REGION Network 97: Step[2046] : Tape Attach Unit HomePos Command
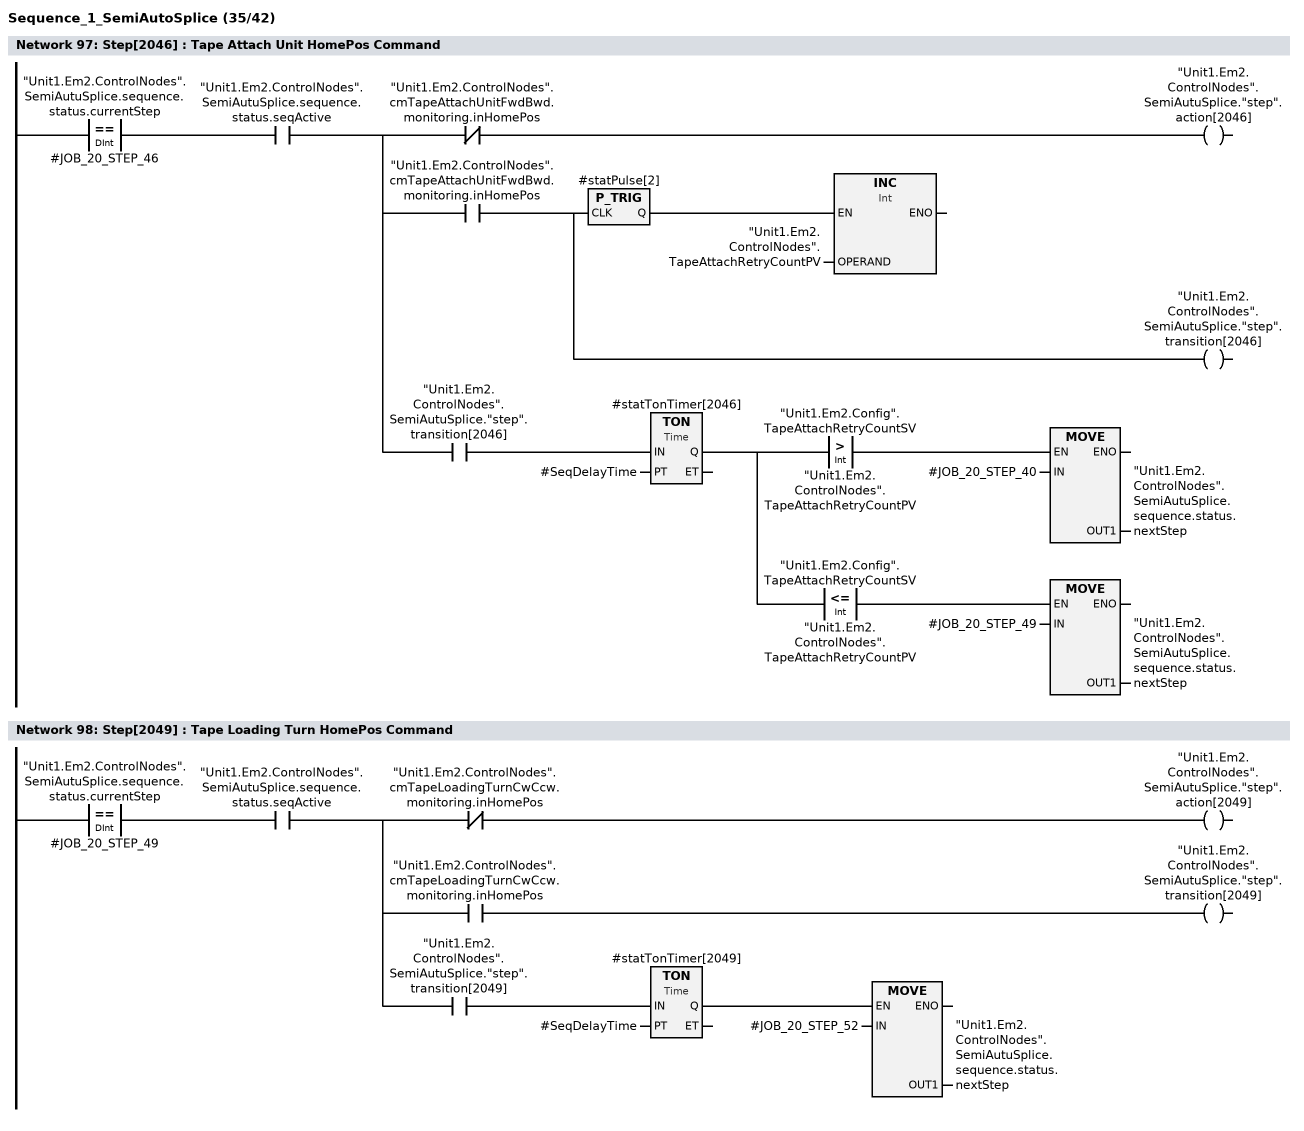
   RUNG wire#powerrail
      { S7_Templates := "SrcType := DInt" } EQ_Contact(in1 := "Unit1.Em2.ControlNodes".SemiAutuSplice.sequence.status.currentStep, in2 := #JOB_20_STEP_46)
      Contact( "Unit1.Em2.ControlNodes".SemiAutuSplice.sequence.status.seqActive )
      wire#w1
      I_Contact( "Unit1.Em2.ControlNodes".cmTapeAttachUnitFwdBwd.monitoring.inHomePos )
      Coil( "Unit1.Em2.ControlNodes".SemiAutuSplice."step".action[2046] )
   END_RUNG
   RUNG wire#w1
      Contact( "Unit1.Em2.ControlNodes".cmTapeAttachUnitFwdBwd.monitoring.inHomePos )
      wire#w2
      P_Trig( #statPulse[2] )
      { S7_Templates := "DestType := Int" } Inc( "Unit1.Em2.ControlNodes".TapeAttachRetryCountPV )
   END_RUNG
   RUNG wire#w2
      Coil( "Unit1.Em2.ControlNodes".SemiAutuSplice."step".transition[2046] )
   END_RUNG
   RUNG wire#w1
      Contact( "Unit1.Em2.ControlNodes".SemiAutuSplice."step".transition[2046] )
      { S7_Templates := "time_type := Time" } #statTonTimer[2046].TON(pt := #SeqDelayTime, et =>)
      wire#w3
      { S7_Templates := "SrcType := Int" } GT_Contact(in1 := "Unit1.Em2.Config".TapeAttachRetryCountSV, in2 := "Unit1.Em2.ControlNodes".TapeAttachRetryCountPV)
      Move(in := #JOB_20_STEP_40, out1 => "Unit1.Em2.ControlNodes".SemiAutuSplice.sequence.status.nextStep)
   END_RUNG
   RUNG wire#w3
      { S7_Templates := "SrcType := Int" } LE_Contact(in1 := "Unit1.Em2.Config".TapeAttachRetryCountSV, in2 := "Unit1.Em2.ControlNodes".TapeAttachRetryCountPV)
      Move(in := #JOB_20_STEP_49, out1 => "Unit1.Em2.ControlNodes".SemiAutuSplice.sequence.status.nextStep)
   END_RUNG
   // the same network as SCL:
   #_w1 := ("Unit1.Em2.ControlNodes".SemiAutuSplice.sequence.status.currentStep = #JOB_20_STEP_46) AND "Unit1.Em2.ControlNodes".SemiAutuSplice.sequence.status.seqActive;
   "Unit1.Em2.ControlNodes".SemiAutuSplice."step".action[2046] := #_w1 AND NOT "Unit1.Em2.ControlNodes".cmTapeAttachUnitFwdBwd.monitoring.inHomePos;
   #_w2 := #_w1 AND "Unit1.Em2.ControlNodes".cmTapeAttachUnitFwdBwd.monitoring.inHomePos;
   #_w3 := #_w2 AND NOT #statPulse[2];   // rising edge
   #statPulse[2] := #_w2;
   IF #_w3 THEN
       "Unit1.Em2.ControlNodes".TapeAttachRetryCountPV := "Unit1.Em2.ControlNodes".TapeAttachRetryCountPV + 1;
   END_IF;
   "Unit1.Em2.ControlNodes".SemiAutuSplice."step".transition[2046] := #_w2;
   #statTonTimer[2046].TON(IN := #_w1 AND "Unit1.Em2.ControlNodes".SemiAutuSplice."step".transition[2046],
                           PT := #SeqDelayTime);
   IF #statTonTimer[2046].Q AND ("Unit1.Em2.Config".TapeAttachRetryCountSV > "Unit1.Em2.ControlNodes".TapeAttachRetryCountPV) THEN
       "Unit1.Em2.ControlNodes".SemiAutuSplice.sequence.status.nextStep := #JOB_20_STEP_40;
   END_IF;
   IF #statTonTimer[2046].Q AND ("Unit1.Em2.Config".TapeAttachRetryCountSV <= "Unit1.Em2.ControlNodes".TapeAttachRetryCountPV) THEN
       "Unit1.Em2.ControlNodes".SemiAutuSplice.sequence.status.nextStep := #JOB_20_STEP_49;
   END_IF;
END_REGION

REGION Network 98: Step[2049] : Tape Loading Turn HomePos Command
   RUNG wire#powerrail
      { S7_Templates := "SrcType := DInt" } EQ_Contact(in1 := "Unit1.Em2.ControlNodes".SemiAutuSplice.sequence.status.currentStep, in2 := #JOB_20_STEP_49)
      Contact( "Unit1.Em2.ControlNodes".SemiAutuSplice.sequence.status.seqActive )
      wire#w1
      I_Contact( "Unit1.Em2.ControlNodes".cmTapeLoadingTurnCwCcw.monitoring.inHomePos )
      Coil( "Unit1.Em2.ControlNodes".SemiAutuSplice."step".action[2049] )
   END_RUNG
   RUNG wire#w1
      Contact( "Unit1.Em2.ControlNodes".cmTapeLoadingTurnCwCcw.monitoring.inHomePos )
      Coil( "Unit1.Em2.ControlNodes".SemiAutuSplice."step".transition[2049] )
   END_RUNG
   RUNG wire#w1
      Contact( "Unit1.Em2.ControlNodes".SemiAutuSplice."step".transition[2049] )
      { S7_Templates := "time_type := Time" } #statTonTimer[2049].TON(pt := #SeqDelayTime, et =>)
      Move(in := #JOB_20_STEP_52, out1 => "Unit1.Em2.ControlNodes".SemiAutuSplice.sequence.status.nextStep)
   END_RUNG
   // the same network as SCL:
   #_w1 := ("Unit1.Em2.ControlNodes".SemiAutuSplice.sequence.status.currentStep = #JOB_20_STEP_49) AND "Unit1.Em2.ControlNodes".SemiAutuSplice.sequence.status.seqActive;
   "Unit1.Em2.ControlNodes".SemiAutuSplice."step".action[2049] := #_w1 AND NOT "Unit1.Em2.ControlNodes".cmTapeLoadingTurnCwCcw.monitoring.inHomePos;
   "Unit1.Em2.ControlNodes".SemiAutuSplice."step".transition[2049] := #_w1 AND "Unit1.Em2.ControlNodes".cmTapeLoadingTurnCwCcw.monitoring.inHomePos;
   #statTonTimer[2049].TON(IN := #_w1 AND "Unit1.Em2.ControlNodes".SemiAutuSplice."step".transition[2049],
                           PT := #SeqDelayTime);
   IF #statTonTimer[2049].Q THEN
       "Unit1.Em2.ControlNodes".SemiAutuSplice.sequence.status.nextStep := #JOB_20_STEP_52;
   END_IF;
END_REGION

REGION Network 99: Step[2052] : Uw Semi Splicer Vacuum Top & Uw Semi Splicer Vacuum Bottom HomePos Command
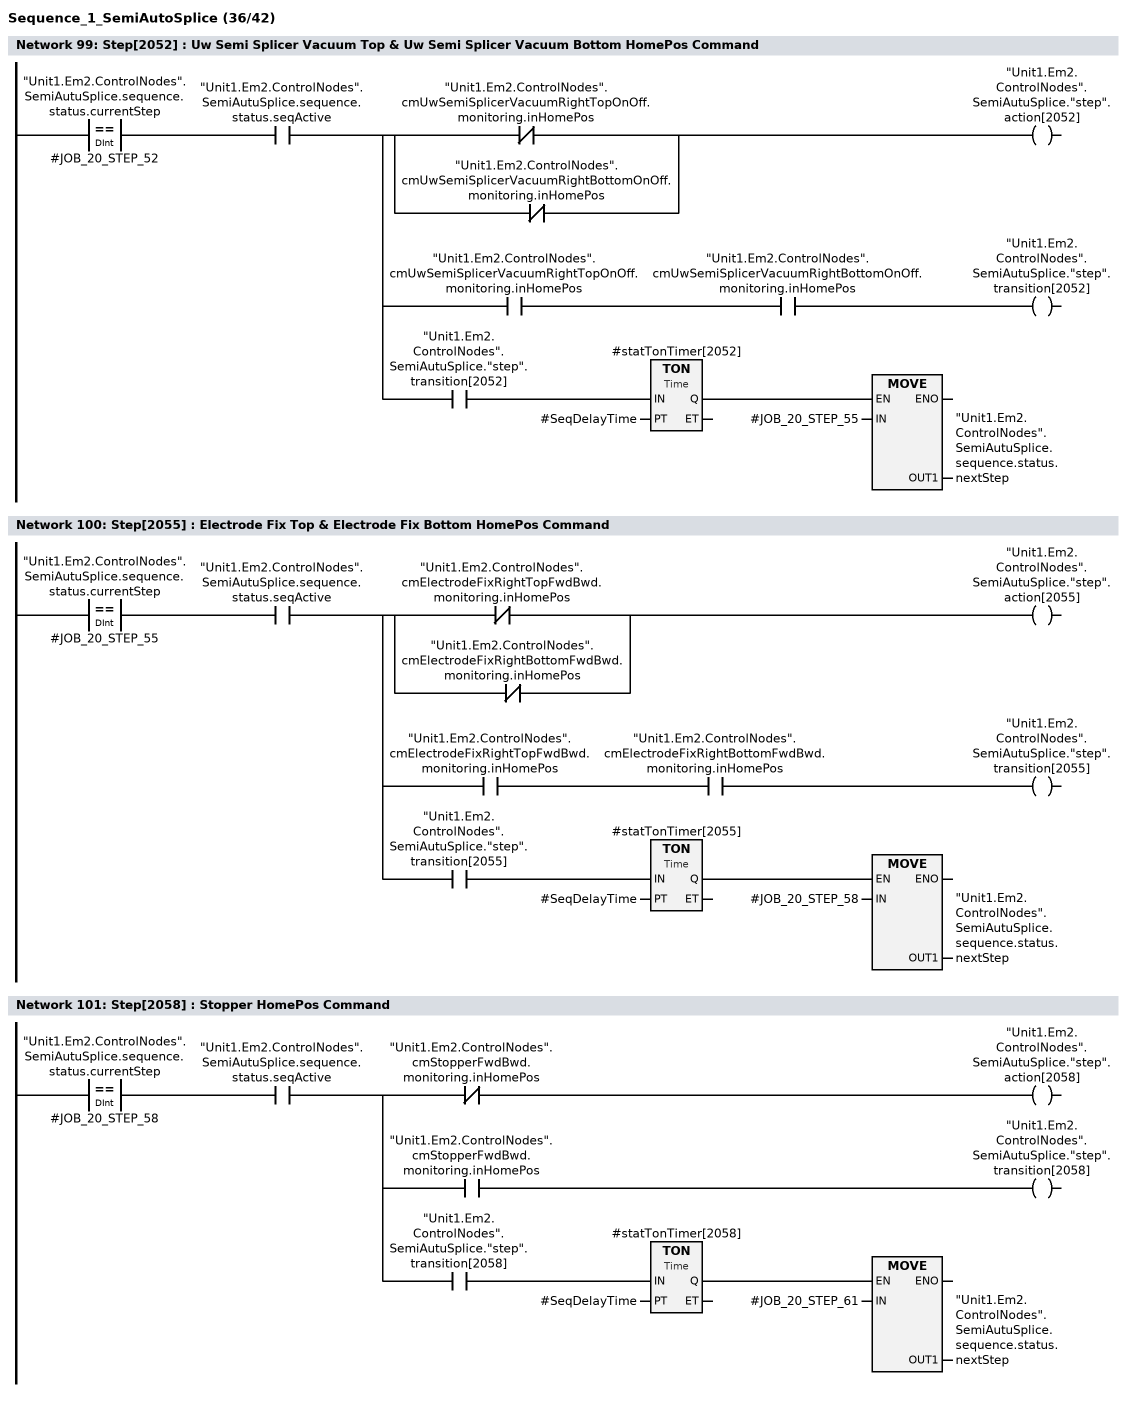
   RUNG wire#powerrail
      { S7_Templates := "SrcType := DInt" } EQ_Contact(in1 := "Unit1.Em2.ControlNodes".SemiAutuSplice.sequence.status.currentStep, in2 := #JOB_20_STEP_52)
      Contact( "Unit1.Em2.ControlNodes".SemiAutuSplice.sequence.status.seqActive )
      wire#w1
      I_Contact( "Unit1.Em2.ControlNodes".cmUwSemiSplicerVacuumRightTopOnOff.monitoring.inHomePos )
      wire#w2
      Coil( "Unit1.Em2.ControlNodes".SemiAutuSplice."step".action[2052] )
   END_RUNG
   RUNG wire#w1
      I_Contact( "Unit1.Em2.ControlNodes".cmUwSemiSplicerVacuumRightBottomOnOff.monitoring.inHomePos )
   END_RUNG wire#w2
   RUNG wire#w1
      Contact( "Unit1.Em2.ControlNodes".cmUwSemiSplicerVacuumRightTopOnOff.monitoring.inHomePos )
      Contact( "Unit1.Em2.ControlNodes".cmUwSemiSplicerVacuumRightBottomOnOff.monitoring.inHomePos )
      Coil( "Unit1.Em2.ControlNodes".SemiAutuSplice."step".transition[2052] )
   END_RUNG
   RUNG wire#w1
      Contact( "Unit1.Em2.ControlNodes".SemiAutuSplice."step".transition[2052] )
      { S7_Templates := "time_type := Time" } #statTonTimer[2052].TON(pt := #SeqDelayTime, et =>)
      Move(in := #JOB_20_STEP_55, out1 => "Unit1.Em2.ControlNodes".SemiAutuSplice.sequence.status.nextStep)
   END_RUNG
   // the same network as SCL:
   #_w1 := ("Unit1.Em2.ControlNodes".SemiAutuSplice.sequence.status.currentStep = #JOB_20_STEP_52) AND "Unit1.Em2.ControlNodes".SemiAutuSplice.sequence.status.seqActive;
   "Unit1.Em2.ControlNodes".SemiAutuSplice."step".action[2052] := #_w1 AND (NOT "Unit1.Em2.ControlNodes".cmUwSemiSplicerVacuumRightTopOnOff.monitoring.inHomePos OR NOT "Unit1.Em2.ControlNodes".cmUwSemiSplicerVacuumRightBottomOnOff.monitoring.inHomePos);
   "Unit1.Em2.ControlNodes".SemiAutuSplice."step".transition[2052] := #_w1 AND "Unit1.Em2.ControlNodes".cmUwSemiSplicerVacuumRightTopOnOff.monitoring.inHomePos AND "Unit1.Em2.ControlNodes".cmUwSemiSplicerVacuumRightBottomOnOff.monitoring.inHomePos;
   #statTonTimer[2052].TON(IN := #_w1 AND "Unit1.Em2.ControlNodes".SemiAutuSplice."step".transition[2052],
                           PT := #SeqDelayTime);
   IF #statTonTimer[2052].Q THEN
       "Unit1.Em2.ControlNodes".SemiAutuSplice.sequence.status.nextStep := #JOB_20_STEP_55;
   END_IF;
END_REGION

REGION Network 100: Step[2055] : Electrode Fix Top & Electrode Fix Bottom HomePos Command
   RUNG wire#powerrail
      { S7_Templates := "SrcType := DInt" } EQ_Contact(in1 := "Unit1.Em2.ControlNodes".SemiAutuSplice.sequence.status.currentStep, in2 := #JOB_20_STEP_55)
      Contact( "Unit1.Em2.ControlNodes".SemiAutuSplice.sequence.status.seqActive )
      wire#w1
      I_Contact( "Unit1.Em2.ControlNodes".cmElectrodeFixRightTopFwdBwd.monitoring.inHomePos )
      wire#w2
      Coil( "Unit1.Em2.ControlNodes".SemiAutuSplice."step".action[2055] )
   END_RUNG
   RUNG wire#w1
      I_Contact( "Unit1.Em2.ControlNodes".cmElectrodeFixRightBottomFwdBwd.monitoring.inHomePos )
   END_RUNG wire#w2
   RUNG wire#w1
      Contact( "Unit1.Em2.ControlNodes".cmElectrodeFixRightTopFwdBwd.monitoring.inHomePos )
      Contact( "Unit1.Em2.ControlNodes".cmElectrodeFixRightBottomFwdBwd.monitoring.inHomePos )
      Coil( "Unit1.Em2.ControlNodes".SemiAutuSplice."step".transition[2055] )
   END_RUNG
   RUNG wire#w1
      Contact( "Unit1.Em2.ControlNodes".SemiAutuSplice."step".transition[2055] )
      { S7_Templates := "time_type := Time" } #statTonTimer[2055].TON(pt := #SeqDelayTime, et =>)
      Move(in := #JOB_20_STEP_58, out1 => "Unit1.Em2.ControlNodes".SemiAutuSplice.sequence.status.nextStep)
   END_RUNG
   // the same network as SCL:
   #_w1 := ("Unit1.Em2.ControlNodes".SemiAutuSplice.sequence.status.currentStep = #JOB_20_STEP_55) AND "Unit1.Em2.ControlNodes".SemiAutuSplice.sequence.status.seqActive;
   "Unit1.Em2.ControlNodes".SemiAutuSplice."step".action[2055] := #_w1 AND (NOT "Unit1.Em2.ControlNodes".cmElectrodeFixRightTopFwdBwd.monitoring.inHomePos OR NOT "Unit1.Em2.ControlNodes".cmElectrodeFixRightBottomFwdBwd.monitoring.inHomePos);
   "Unit1.Em2.ControlNodes".SemiAutuSplice."step".transition[2055] := #_w1 AND "Unit1.Em2.ControlNodes".cmElectrodeFixRightTopFwdBwd.monitoring.inHomePos AND "Unit1.Em2.ControlNodes".cmElectrodeFixRightBottomFwdBwd.monitoring.inHomePos;
   #statTonTimer[2055].TON(IN := #_w1 AND "Unit1.Em2.ControlNodes".SemiAutuSplice."step".transition[2055],
                           PT := #SeqDelayTime);
   IF #statTonTimer[2055].Q THEN
       "Unit1.Em2.ControlNodes".SemiAutuSplice.sequence.status.nextStep := #JOB_20_STEP_58;
   END_IF;
END_REGION

REGION Network 101: Step[2058] : Stopper HomePos Command
   RUNG wire#powerrail
      { S7_Templates := "SrcType := DInt" } EQ_Contact(in1 := "Unit1.Em2.ControlNodes".SemiAutuSplice.sequence.status.currentStep, in2 := #JOB_20_STEP_58)
      Contact( "Unit1.Em2.ControlNodes".SemiAutuSplice.sequence.status.seqActive )
      wire#w1
      I_Contact( "Unit1.Em2.ControlNodes".cmStopperFwdBwd.monitoring.inHomePos )
      Coil( "Unit1.Em2.ControlNodes".SemiAutuSplice."step".action[2058] )
   END_RUNG
   RUNG wire#w1
      Contact( "Unit1.Em2.ControlNodes".cmStopperFwdBwd.monitoring.inHomePos )
      Coil( "Unit1.Em2.ControlNodes".SemiAutuSplice."step".transition[2058] )
   END_RUNG
   RUNG wire#w1
      Contact( "Unit1.Em2.ControlNodes".SemiAutuSplice."step".transition[2058] )
      { S7_Templates := "time_type := Time" } #statTonTimer[2058].TON(pt := #SeqDelayTime, et =>)
      Move(in := #JOB_20_STEP_61, out1 => "Unit1.Em2.ControlNodes".SemiAutuSplice.sequence.status.nextStep)
   END_RUNG
   // the same network as SCL:
   #_w1 := ("Unit1.Em2.ControlNodes".SemiAutuSplice.sequence.status.currentStep = #JOB_20_STEP_58) AND "Unit1.Em2.ControlNodes".SemiAutuSplice.sequence.status.seqActive;
   "Unit1.Em2.ControlNodes".SemiAutuSplice."step".action[2058] := #_w1 AND NOT "Unit1.Em2.ControlNodes".cmStopperFwdBwd.monitoring.inHomePos;
   "Unit1.Em2.ControlNodes".SemiAutuSplice."step".transition[2058] := #_w1 AND "Unit1.Em2.ControlNodes".cmStopperFwdBwd.monitoring.inHomePos;
   #statTonTimer[2058].TON(IN := #_w1 AND "Unit1.Em2.ControlNodes".SemiAutuSplice."step".transition[2058],
                           PT := #SeqDelayTime);
   IF #statTonTimer[2058].Q THEN
       "Unit1.Em2.ControlNodes".SemiAutuSplice.sequence.status.nextStep := #JOB_20_STEP_61;
   END_IF;
END_REGION

REGION Network 102: Step[2061] : EM Link Change Check
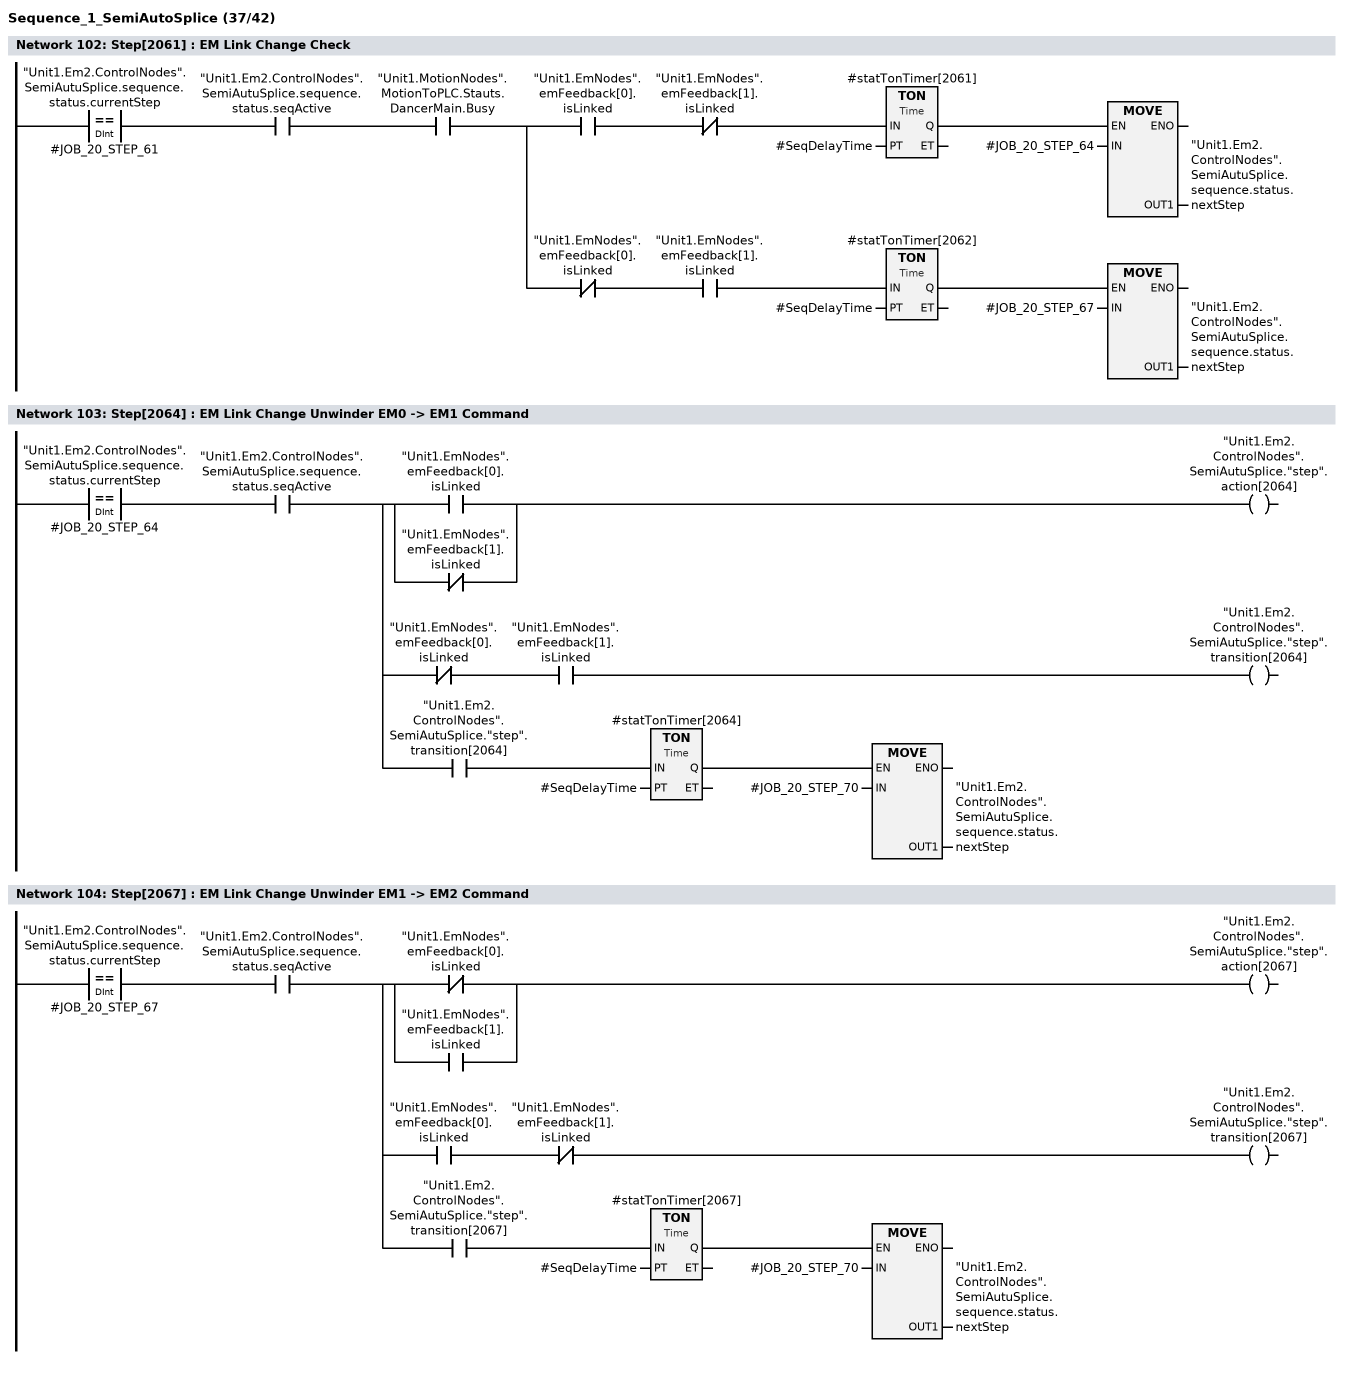
   RUNG wire#powerrail
      { S7_Templates := "SrcType := DInt" } EQ_Contact(in1 := "Unit1.Em2.ControlNodes".SemiAutuSplice.sequence.status.currentStep, in2 := #JOB_20_STEP_61)
      Contact( "Unit1.Em2.ControlNodes".SemiAutuSplice.sequence.status.seqActive )
      Contact( "Unit1.MotionNodes".MotionToPLC.Stauts.DancerMain.Busy )
      wire#w1
      Contact( "Unit1.EmNodes".emFeedback[0].isLinked )
      I_Contact( "Unit1.EmNodes".emFeedback[1].isLinked )
      { S7_Templates := "time_type := Time" } #statTonTimer[2061].TON(pt := #SeqDelayTime, et =>)
      Move(in := #JOB_20_STEP_64, out1 => "Unit1.Em2.ControlNodes".SemiAutuSplice.sequence.status.nextStep)
   END_RUNG
   RUNG wire#w1
      I_Contact( "Unit1.EmNodes".emFeedback[0].isLinked )
      Contact( "Unit1.EmNodes".emFeedback[1].isLinked )
      { S7_Templates := "time_type := Time" } #statTonTimer[2062].TON(pt := #SeqDelayTime, et =>)
      Move(in := #JOB_20_STEP_67, out1 => "Unit1.Em2.ControlNodes".SemiAutuSplice.sequence.status.nextStep)
   END_RUNG
   // the same network as SCL:
   #_w1 := ("Unit1.Em2.ControlNodes".SemiAutuSplice.sequence.status.currentStep = #JOB_20_STEP_61) AND "Unit1.Em2.ControlNodes".SemiAutuSplice.sequence.status.seqActive AND "Unit1.MotionNodes".MotionToPLC.Stauts.DancerMain.Busy;
   #statTonTimer[2061].TON(IN := #_w1 AND "Unit1.EmNodes".emFeedback[0].isLinked AND NOT "Unit1.EmNodes".emFeedback[1].isLinked,
                           PT := #SeqDelayTime);
   IF #statTonTimer[2061].Q THEN
       "Unit1.Em2.ControlNodes".SemiAutuSplice.sequence.status.nextStep := #JOB_20_STEP_64;
   END_IF;
   #statTonTimer[2062].TON(IN := #_w1 AND NOT "Unit1.EmNodes".emFeedback[0].isLinked AND "Unit1.EmNodes".emFeedback[1].isLinked,
                           PT := #SeqDelayTime);
   IF #statTonTimer[2062].Q THEN
       "Unit1.Em2.ControlNodes".SemiAutuSplice.sequence.status.nextStep := #JOB_20_STEP_67;
   END_IF;
END_REGION

REGION Network 103: Step[2064] : EM Link Change Unwinder EM0 -> EM1 Command
   RUNG wire#powerrail
      { S7_Templates := "SrcType := DInt" } EQ_Contact(in1 := "Unit1.Em2.ControlNodes".SemiAutuSplice.sequence.status.currentStep, in2 := #JOB_20_STEP_64)
      Contact( "Unit1.Em2.ControlNodes".SemiAutuSplice.sequence.status.seqActive )
      wire#w1
      Contact( "Unit1.EmNodes".emFeedback[0].isLinked )
      wire#w2
      Coil( "Unit1.Em2.ControlNodes".SemiAutuSplice."step".action[2064] )
   END_RUNG
   RUNG wire#w1
      I_Contact( "Unit1.EmNodes".emFeedback[1].isLinked )
   END_RUNG wire#w2
   RUNG wire#w1
      I_Contact( "Unit1.EmNodes".emFeedback[0].isLinked )
      Contact( "Unit1.EmNodes".emFeedback[1].isLinked )
      Coil( "Unit1.Em2.ControlNodes".SemiAutuSplice."step".transition[2064] )
   END_RUNG
   RUNG wire#w1
      Contact( "Unit1.Em2.ControlNodes".SemiAutuSplice."step".transition[2064] )
      { S7_Templates := "time_type := Time" } #statTonTimer[2064].TON(pt := #SeqDelayTime, et =>)
      Move(in := #JOB_20_STEP_70, out1 => "Unit1.Em2.ControlNodes".SemiAutuSplice.sequence.status.nextStep)
   END_RUNG
   // the same network as SCL:
   #_w1 := ("Unit1.Em2.ControlNodes".SemiAutuSplice.sequence.status.currentStep = #JOB_20_STEP_64) AND "Unit1.Em2.ControlNodes".SemiAutuSplice.sequence.status.seqActive;
   "Unit1.Em2.ControlNodes".SemiAutuSplice."step".action[2064] := #_w1 AND ("Unit1.EmNodes".emFeedback[0].isLinked OR NOT "Unit1.EmNodes".emFeedback[1].isLinked);
   "Unit1.Em2.ControlNodes".SemiAutuSplice."step".transition[2064] := #_w1 AND NOT "Unit1.EmNodes".emFeedback[0].isLinked AND "Unit1.EmNodes".emFeedback[1].isLinked;
   #statTonTimer[2064].TON(IN := #_w1 AND "Unit1.Em2.ControlNodes".SemiAutuSplice."step".transition[2064],
                           PT := #SeqDelayTime);
   IF #statTonTimer[2064].Q THEN
       "Unit1.Em2.ControlNodes".SemiAutuSplice.sequence.status.nextStep := #JOB_20_STEP_70;
   END_IF;
END_REGION

REGION Network 104: Step[2067] : EM Link Change Unwinder EM1 -> EM2 Command
   RUNG wire#powerrail
      { S7_Templates := "SrcType := DInt" } EQ_Contact(in1 := "Unit1.Em2.ControlNodes".SemiAutuSplice.sequence.status.currentStep, in2 := #JOB_20_STEP_67)
      Contact( "Unit1.Em2.ControlNodes".SemiAutuSplice.sequence.status.seqActive )
      wire#w1
      I_Contact( "Unit1.EmNodes".emFeedback[0].isLinked )
      wire#w2
      Coil( "Unit1.Em2.ControlNodes".SemiAutuSplice."step".action[2067] )
   END_RUNG
   RUNG wire#w1
      Contact( "Unit1.EmNodes".emFeedback[1].isLinked )
   END_RUNG wire#w2
   RUNG wire#w1
      Contact( "Unit1.EmNodes".emFeedback[0].isLinked )
      I_Contact( "Unit1.EmNodes".emFeedback[1].isLinked )
      Coil( "Unit1.Em2.ControlNodes".SemiAutuSplice."step".transition[2067] )
   END_RUNG
   RUNG wire#w1
      Contact( "Unit1.Em2.ControlNodes".SemiAutuSplice."step".transition[2067] )
      { S7_Templates := "time_type := Time" } #statTonTimer[2067].TON(pt := #SeqDelayTime, et =>)
      Move(in := #JOB_20_STEP_70, out1 => "Unit1.Em2.ControlNodes".SemiAutuSplice.sequence.status.nextStep)
   END_RUNG
   // the same network as SCL:
   #_w1 := ("Unit1.Em2.ControlNodes".SemiAutuSplice.sequence.status.currentStep = #JOB_20_STEP_67) AND "Unit1.Em2.ControlNodes".SemiAutuSplice.sequence.status.seqActive;
   "Unit1.Em2.ControlNodes".SemiAutuSplice."step".action[2067] := #_w1 AND (NOT "Unit1.EmNodes".emFeedback[0].isLinked OR "Unit1.EmNodes".emFeedback[1].isLinked);
   "Unit1.Em2.ControlNodes".SemiAutuSplice."step".transition[2067] := #_w1 AND "Unit1.EmNodes".emFeedback[0].isLinked AND NOT "Unit1.EmNodes".emFeedback[1].isLinked;
   #statTonTimer[2067].TON(IN := #_w1 AND "Unit1.Em2.ControlNodes".SemiAutuSplice."step".transition[2067],
                           PT := #SeqDelayTime);
   IF #statTonTimer[2067].Q THEN
       "Unit1.Em2.ControlNodes".SemiAutuSplice.sequence.status.nextStep := #JOB_20_STEP_70;
   END_IF;
END_REGION

REGION Network 105: Step[2070] : EM Link Change Comp
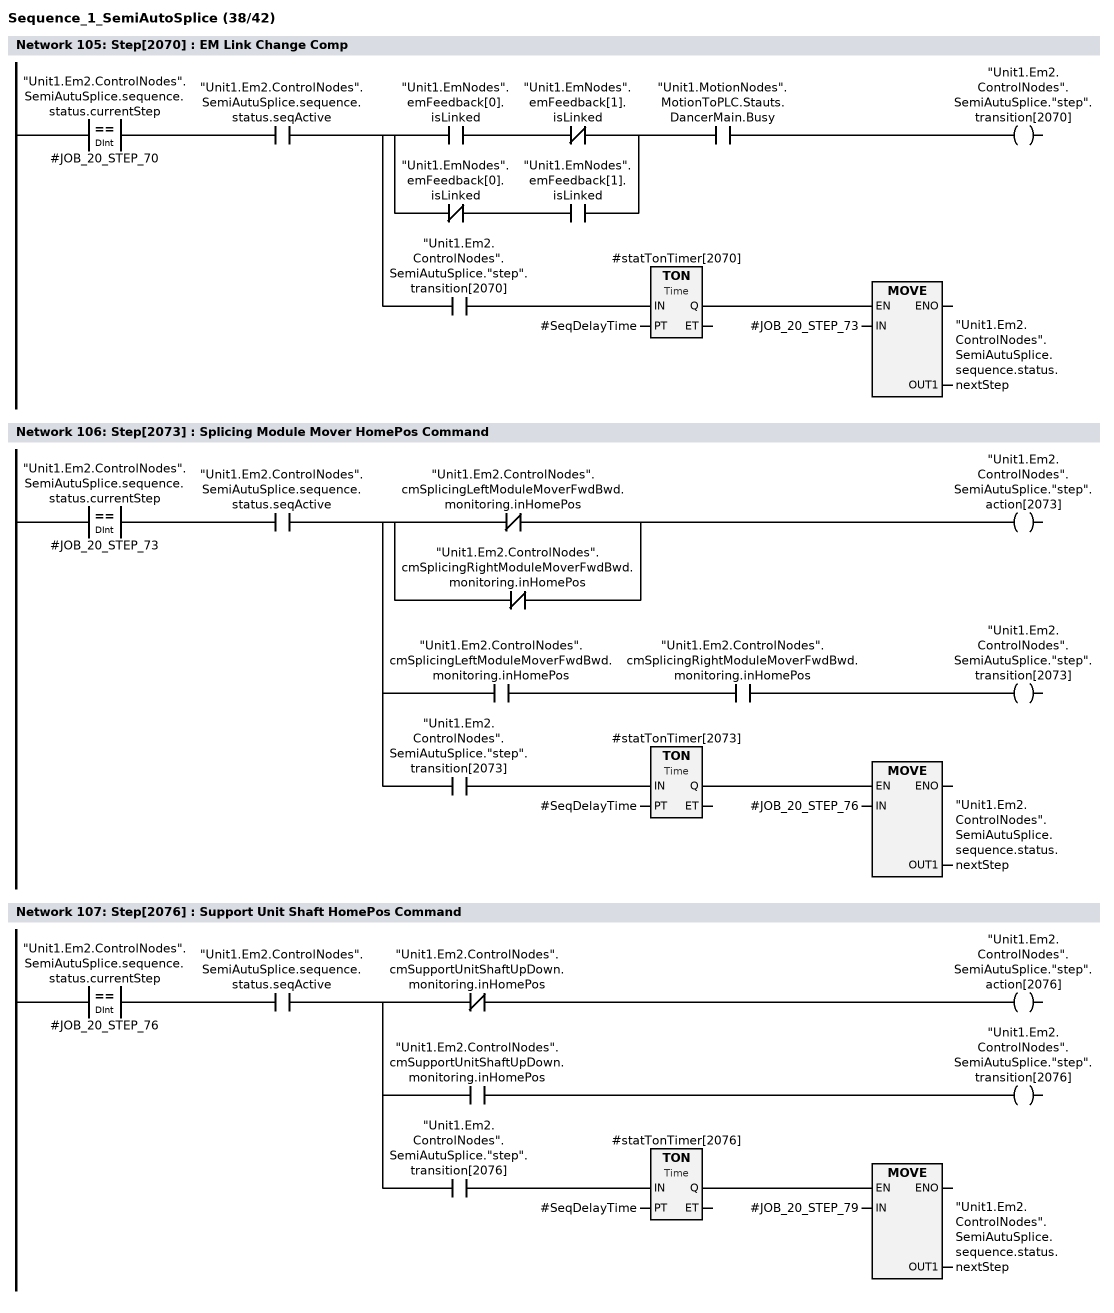
   RUNG wire#powerrail
      { S7_Templates := "SrcType := DInt" } EQ_Contact(in1 := "Unit1.Em2.ControlNodes".SemiAutuSplice.sequence.status.currentStep, in2 := #JOB_20_STEP_70)
      Contact( "Unit1.Em2.ControlNodes".SemiAutuSplice.sequence.status.seqActive )
      wire#w1
      Contact( "Unit1.EmNodes".emFeedback[0].isLinked )
      I_Contact( "Unit1.EmNodes".emFeedback[1].isLinked )
      wire#w2
      Contact( "Unit1.MotionNodes".MotionToPLC.Stauts.DancerMain.Busy )
      Coil( "Unit1.Em2.ControlNodes".SemiAutuSplice."step".transition[2070] )
   END_RUNG
   RUNG wire#w1
      I_Contact( "Unit1.EmNodes".emFeedback[0].isLinked )
      Contact( "Unit1.EmNodes".emFeedback[1].isLinked )
   END_RUNG wire#w2
   RUNG wire#w1
      Contact( "Unit1.Em2.ControlNodes".SemiAutuSplice."step".transition[2070] )
      { S7_Templates := "time_type := Time" } #statTonTimer[2070].TON(pt := #SeqDelayTime, et =>)
      Move(in := #JOB_20_STEP_73, out1 => "Unit1.Em2.ControlNodes".SemiAutuSplice.sequence.status.nextStep)
   END_RUNG
   // the same network as SCL:
   #_w1 := ("Unit1.Em2.ControlNodes".SemiAutuSplice.sequence.status.currentStep = #JOB_20_STEP_70) AND "Unit1.Em2.ControlNodes".SemiAutuSplice.sequence.status.seqActive;
   "Unit1.Em2.ControlNodes".SemiAutuSplice."step".transition[2070] := #_w1 AND (("Unit1.EmNodes".emFeedback[0].isLinked AND NOT "Unit1.EmNodes".emFeedback[1].isLinked) OR (NOT "Unit1.EmNodes".emFeedback[0].isLinked AND "Unit1.EmNodes".emFeedback[1].isLinked)) AND "Unit1.MotionNodes".MotionToPLC.Stauts.DancerMain.Busy;
   #statTonTimer[2070].TON(IN := #_w1 AND "Unit1.Em2.ControlNodes".SemiAutuSplice."step".transition[2070],
                           PT := #SeqDelayTime);
   IF #statTonTimer[2070].Q THEN
       "Unit1.Em2.ControlNodes".SemiAutuSplice.sequence.status.nextStep := #JOB_20_STEP_73;
   END_IF;
END_REGION

REGION Network 106: Step[2073] : Splicing Module Mover HomePos Command
   RUNG wire#powerrail
      { S7_Templates := "SrcType := DInt" } EQ_Contact(in1 := "Unit1.Em2.ControlNodes".SemiAutuSplice.sequence.status.currentStep, in2 := #JOB_20_STEP_73)
      Contact( "Unit1.Em2.ControlNodes".SemiAutuSplice.sequence.status.seqActive )
      wire#w1
      I_Contact( "Unit1.Em2.ControlNodes".cmSplicingLeftModuleMoverFwdBwd.monitoring.inHomePos )
      wire#w2
      Coil( "Unit1.Em2.ControlNodes".SemiAutuSplice."step".action[2073] )
   END_RUNG
   RUNG wire#w1
      I_Contact( "Unit1.Em2.ControlNodes".cmSplicingRightModuleMoverFwdBwd.monitoring.inHomePos )
   END_RUNG wire#w2
   RUNG wire#w1
      Contact( "Unit1.Em2.ControlNodes".cmSplicingLeftModuleMoverFwdBwd.monitoring.inHomePos )
      Contact( "Unit1.Em2.ControlNodes".cmSplicingRightModuleMoverFwdBwd.monitoring.inHomePos )
      Coil( "Unit1.Em2.ControlNodes".SemiAutuSplice."step".transition[2073] )
   END_RUNG
   RUNG wire#w1
      Contact( "Unit1.Em2.ControlNodes".SemiAutuSplice."step".transition[2073] )
      { S7_Templates := "time_type := Time" } #statTonTimer[2073].TON(pt := #SeqDelayTime, et =>)
      Move(in := #JOB_20_STEP_76, out1 => "Unit1.Em2.ControlNodes".SemiAutuSplice.sequence.status.nextStep)
   END_RUNG
   // the same network as SCL:
   #_w1 := ("Unit1.Em2.ControlNodes".SemiAutuSplice.sequence.status.currentStep = #JOB_20_STEP_73) AND "Unit1.Em2.ControlNodes".SemiAutuSplice.sequence.status.seqActive;
   "Unit1.Em2.ControlNodes".SemiAutuSplice."step".action[2073] := #_w1 AND (NOT "Unit1.Em2.ControlNodes".cmSplicingLeftModuleMoverFwdBwd.monitoring.inHomePos OR NOT "Unit1.Em2.ControlNodes".cmSplicingRightModuleMoverFwdBwd.monitoring.inHomePos);
   "Unit1.Em2.ControlNodes".SemiAutuSplice."step".transition[2073] := #_w1 AND "Unit1.Em2.ControlNodes".cmSplicingLeftModuleMoverFwdBwd.monitoring.inHomePos AND "Unit1.Em2.ControlNodes".cmSplicingRightModuleMoverFwdBwd.monitoring.inHomePos;
   #statTonTimer[2073].TON(IN := #_w1 AND "Unit1.Em2.ControlNodes".SemiAutuSplice."step".transition[2073],
                           PT := #SeqDelayTime);
   IF #statTonTimer[2073].Q THEN
       "Unit1.Em2.ControlNodes".SemiAutuSplice.sequence.status.nextStep := #JOB_20_STEP_76;
   END_IF;
END_REGION

REGION Network 107: Step[2076] : Support Unit Shaft HomePos Command
   RUNG wire#powerrail
      { S7_Templates := "SrcType := DInt" } EQ_Contact(in1 := "Unit1.Em2.ControlNodes".SemiAutuSplice.sequence.status.currentStep, in2 := #JOB_20_STEP_76)
      Contact( "Unit1.Em2.ControlNodes".SemiAutuSplice.sequence.status.seqActive )
      wire#w1
      I_Contact( "Unit1.Em2.ControlNodes".cmSupportUnitShaftUpDown.monitoring.inHomePos )
      Coil( "Unit1.Em2.ControlNodes".SemiAutuSplice."step".action[2076] )
   END_RUNG
   RUNG wire#w1
      Contact( "Unit1.Em2.ControlNodes".cmSupportUnitShaftUpDown.monitoring.inHomePos )
      Coil( "Unit1.Em2.ControlNodes".SemiAutuSplice."step".transition[2076] )
   END_RUNG
   RUNG wire#w1
      Contact( "Unit1.Em2.ControlNodes".SemiAutuSplice."step".transition[2076] )
      { S7_Templates := "time_type := Time" } #statTonTimer[2076].TON(pt := #SeqDelayTime, et =>)
      Move(in := #JOB_20_STEP_79, out1 => "Unit1.Em2.ControlNodes".SemiAutuSplice.sequence.status.nextStep)
   END_RUNG
   // the same network as SCL:
   #_w1 := ("Unit1.Em2.ControlNodes".SemiAutuSplice.sequence.status.currentStep = #JOB_20_STEP_76) AND "Unit1.Em2.ControlNodes".SemiAutuSplice.sequence.status.seqActive;
   "Unit1.Em2.ControlNodes".SemiAutuSplice."step".action[2076] := #_w1 AND NOT "Unit1.Em2.ControlNodes".cmSupportUnitShaftUpDown.monitoring.inHomePos;
   "Unit1.Em2.ControlNodes".SemiAutuSplice."step".transition[2076] := #_w1 AND "Unit1.Em2.ControlNodes".cmSupportUnitShaftUpDown.monitoring.inHomePos;
   #statTonTimer[2076].TON(IN := #_w1 AND "Unit1.Em2.ControlNodes".SemiAutuSplice."step".transition[2076],
                           PT := #SeqDelayTime);
   IF #statTonTimer[2076].Q THEN
       "Unit1.Em2.ControlNodes".SemiAutuSplice.sequence.status.nextStep := #JOB_20_STEP_79;
   END_IF;
END_REGION

REGION Network 108: Step[2079] : FrameCover HomePos Command
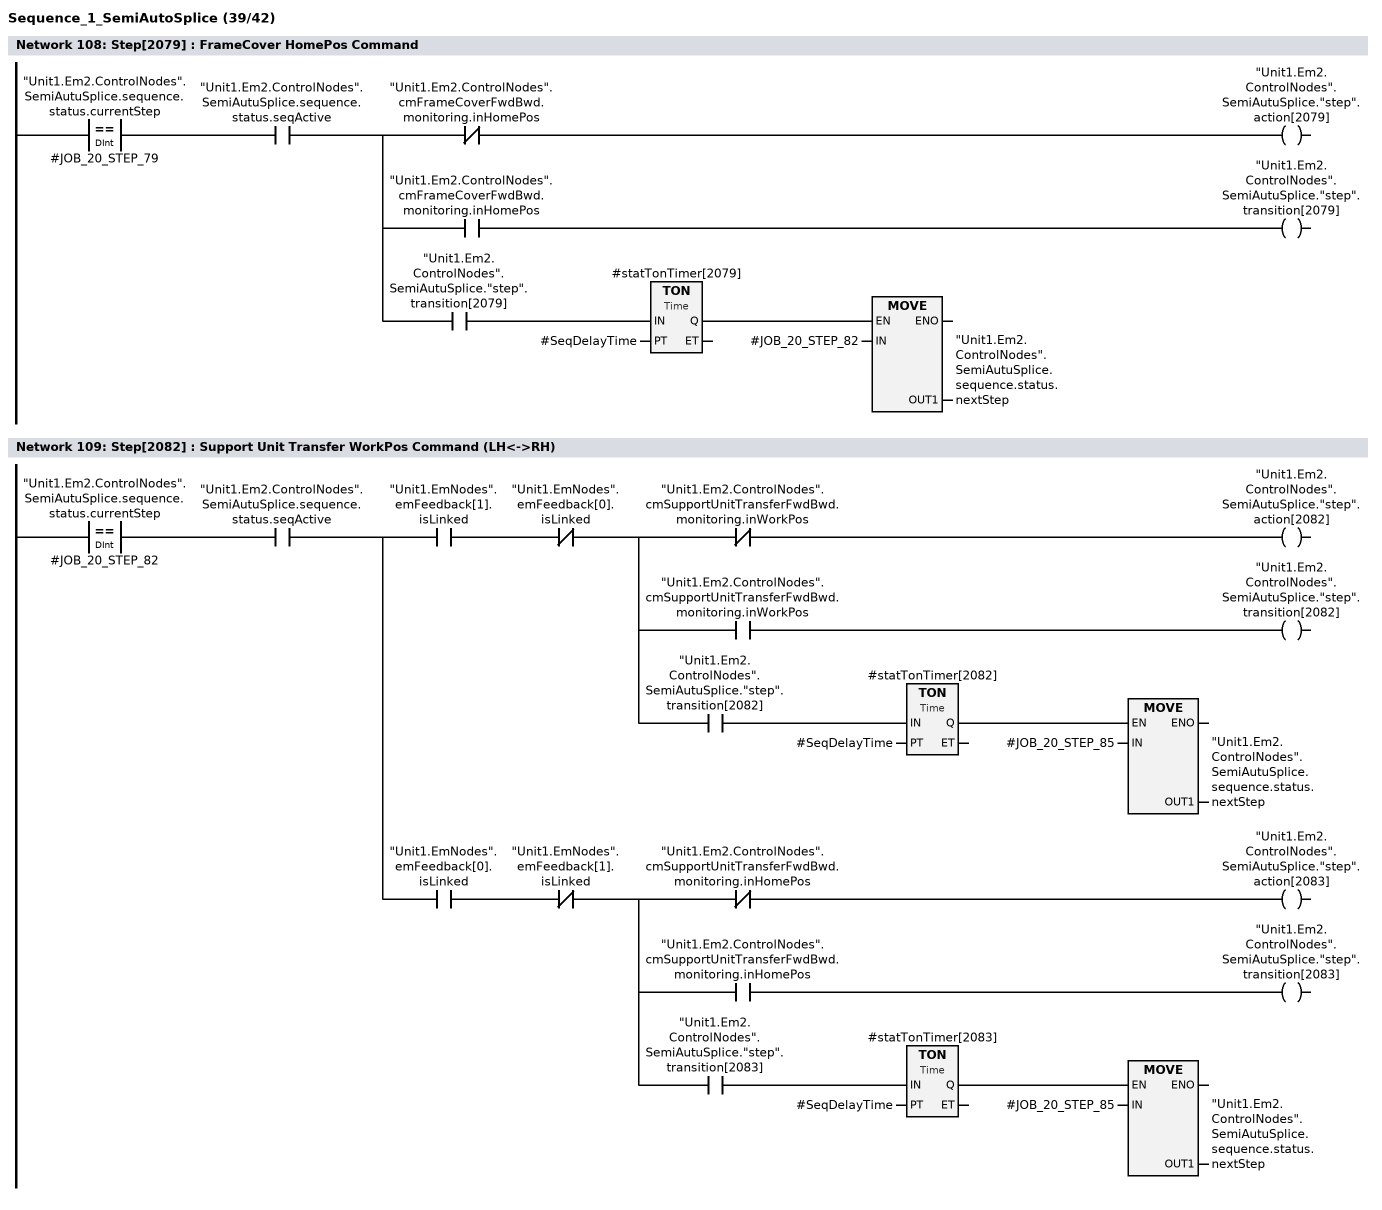
   RUNG wire#powerrail
      { S7_Templates := "SrcType := DInt" } EQ_Contact(in1 := "Unit1.Em2.ControlNodes".SemiAutuSplice.sequence.status.currentStep, in2 := #JOB_20_STEP_79)
      Contact( "Unit1.Em2.ControlNodes".SemiAutuSplice.sequence.status.seqActive )
      wire#w1
      I_Contact( "Unit1.Em2.ControlNodes".cmFrameCoverFwdBwd.monitoring.inHomePos )
      Coil( "Unit1.Em2.ControlNodes".SemiAutuSplice."step".action[2079] )
   END_RUNG
   RUNG wire#w1
      Contact( "Unit1.Em2.ControlNodes".cmFrameCoverFwdBwd.monitoring.inHomePos )
      Coil( "Unit1.Em2.ControlNodes".SemiAutuSplice."step".transition[2079] )
   END_RUNG
   RUNG wire#w1
      Contact( "Unit1.Em2.ControlNodes".SemiAutuSplice."step".transition[2079] )
      { S7_Templates := "time_type := Time" } #statTonTimer[2079].TON(pt := #SeqDelayTime, et =>)
      Move(in := #JOB_20_STEP_82, out1 => "Unit1.Em2.ControlNodes".SemiAutuSplice.sequence.status.nextStep)
   END_RUNG
   // the same network as SCL:
   #_w1 := ("Unit1.Em2.ControlNodes".SemiAutuSplice.sequence.status.currentStep = #JOB_20_STEP_79) AND "Unit1.Em2.ControlNodes".SemiAutuSplice.sequence.status.seqActive;
   "Unit1.Em2.ControlNodes".SemiAutuSplice."step".action[2079] := #_w1 AND NOT "Unit1.Em2.ControlNodes".cmFrameCoverFwdBwd.monitoring.inHomePos;
   "Unit1.Em2.ControlNodes".SemiAutuSplice."step".transition[2079] := #_w1 AND "Unit1.Em2.ControlNodes".cmFrameCoverFwdBwd.monitoring.inHomePos;
   #statTonTimer[2079].TON(IN := #_w1 AND "Unit1.Em2.ControlNodes".SemiAutuSplice."step".transition[2079],
                           PT := #SeqDelayTime);
   IF #statTonTimer[2079].Q THEN
       "Unit1.Em2.ControlNodes".SemiAutuSplice.sequence.status.nextStep := #JOB_20_STEP_82;
   END_IF;
END_REGION

REGION Network 109: Step[2082] : Support Unit Transfer WorkPos Command (LH<->RH)
   RUNG wire#powerrail
      { S7_Templates := "SrcType := DInt" } EQ_Contact(in1 := "Unit1.Em2.ControlNodes".SemiAutuSplice.sequence.status.currentStep, in2 := #JOB_20_STEP_82)
      Contact( "Unit1.Em2.ControlNodes".SemiAutuSplice.sequence.status.seqActive )
      wire#w1
      Contact( "Unit1.EmNodes".emFeedback[1].isLinked )
      I_Contact( "Unit1.EmNodes".emFeedback[0].isLinked )
      wire#w2
      I_Contact( "Unit1.Em2.ControlNodes".cmSupportUnitTransferFwdBwd.monitoring.inWorkPos )
      Coil( "Unit1.Em2.ControlNodes".SemiAutuSplice."step".action[2082] )
   END_RUNG
   RUNG wire#w2
      Contact( "Unit1.Em2.ControlNodes".cmSupportUnitTransferFwdBwd.monitoring.inWorkPos )
      Coil( "Unit1.Em2.ControlNodes".SemiAutuSplice."step".transition[2082] )
   END_RUNG
   RUNG wire#w2
      Contact( "Unit1.Em2.ControlNodes".SemiAutuSplice."step".transition[2082] )
      { S7_Templates := "time_type := Time" } #statTonTimer[2082].TON(pt := #SeqDelayTime, et =>)
      Move(in := #JOB_20_STEP_85, out1 => "Unit1.Em2.ControlNodes".SemiAutuSplice.sequence.status.nextStep)
   END_RUNG
   RUNG wire#w1
      Contact( "Unit1.EmNodes".emFeedback[0].isLinked )
      I_Contact( "Unit1.EmNodes".emFeedback[1].isLinked )
      wire#w3
      I_Contact( "Unit1.Em2.ControlNodes".cmSupportUnitTransferFwdBwd.monitoring.inHomePos )
      Coil( "Unit1.Em2.ControlNodes".SemiAutuSplice."step".action[2083] )
   END_RUNG
   RUNG wire#w3
      Contact( "Unit1.Em2.ControlNodes".cmSupportUnitTransferFwdBwd.monitoring.inHomePos )
      Coil( "Unit1.Em2.ControlNodes".SemiAutuSplice."step".transition[2083] )
   END_RUNG
   RUNG wire#w3
      Contact( "Unit1.Em2.ControlNodes".SemiAutuSplice."step".transition[2083] )
      { S7_Templates := "time_type := Time" } #statTonTimer[2083].TON(pt := #SeqDelayTime, et =>)
      Move(in := #JOB_20_STEP_85, out1 => "Unit1.Em2.ControlNodes".SemiAutuSplice.sequence.status.nextStep)
   END_RUNG
   // the same network as SCL:
   #_w1 := ("Unit1.Em2.ControlNodes".SemiAutuSplice.sequence.status.currentStep = #JOB_20_STEP_82) AND "Unit1.Em2.ControlNodes".SemiAutuSplice.sequence.status.seqActive;
   #_w2 := #_w1 AND "Unit1.EmNodes".emFeedback[1].isLinked AND NOT "Unit1.EmNodes".emFeedback[0].isLinked;
   "Unit1.Em2.ControlNodes".SemiAutuSplice."step".action[2082] := #_w2 AND NOT "Unit1.Em2.ControlNodes".cmSupportUnitTransferFwdBwd.monitoring.inWorkPos;
   "Unit1.Em2.ControlNodes".SemiAutuSplice."step".transition[2082] := #_w2 AND "Unit1.Em2.ControlNodes".cmSupportUnitTransferFwdBwd.monitoring.inWorkPos;
   #statTonTimer[2082].TON(IN := #_w2 AND "Unit1.Em2.ControlNodes".SemiAutuSplice."step".transition[2082],
                           PT := #SeqDelayTime);
   IF #statTonTimer[2082].Q THEN
       "Unit1.Em2.ControlNodes".SemiAutuSplice.sequence.status.nextStep := #JOB_20_STEP_85;
   END_IF;
   #_w3 := #_w1 AND "Unit1.EmNodes".emFeedback[0].isLinked AND NOT "Unit1.EmNodes".emFeedback[1].isLinked;
   "Unit1.Em2.ControlNodes".SemiAutuSplice."step".action[2083] := #_w3 AND NOT "Unit1.Em2.ControlNodes".cmSupportUnitTransferFwdBwd.monitoring.inHomePos;
   "Unit1.Em2.ControlNodes".SemiAutuSplice."step".transition[2083] := #_w3 AND "Unit1.Em2.ControlNodes".cmSupportUnitTransferFwdBwd.monitoring.inHomePos;
   #statTonTimer[2083].TON(IN := #_w3 AND "Unit1.Em2.ControlNodes".SemiAutuSplice."step".transition[2083],
                           PT := #SeqDelayTime);
   IF #statTonTimer[2083].Q THEN
       "Unit1.Em2.ControlNodes".SemiAutuSplice.sequence.status.nextStep := #JOB_20_STEP_85;
   END_IF;
END_REGION

REGION Network 110: Step[2085] : FrameCover WorkPos Command
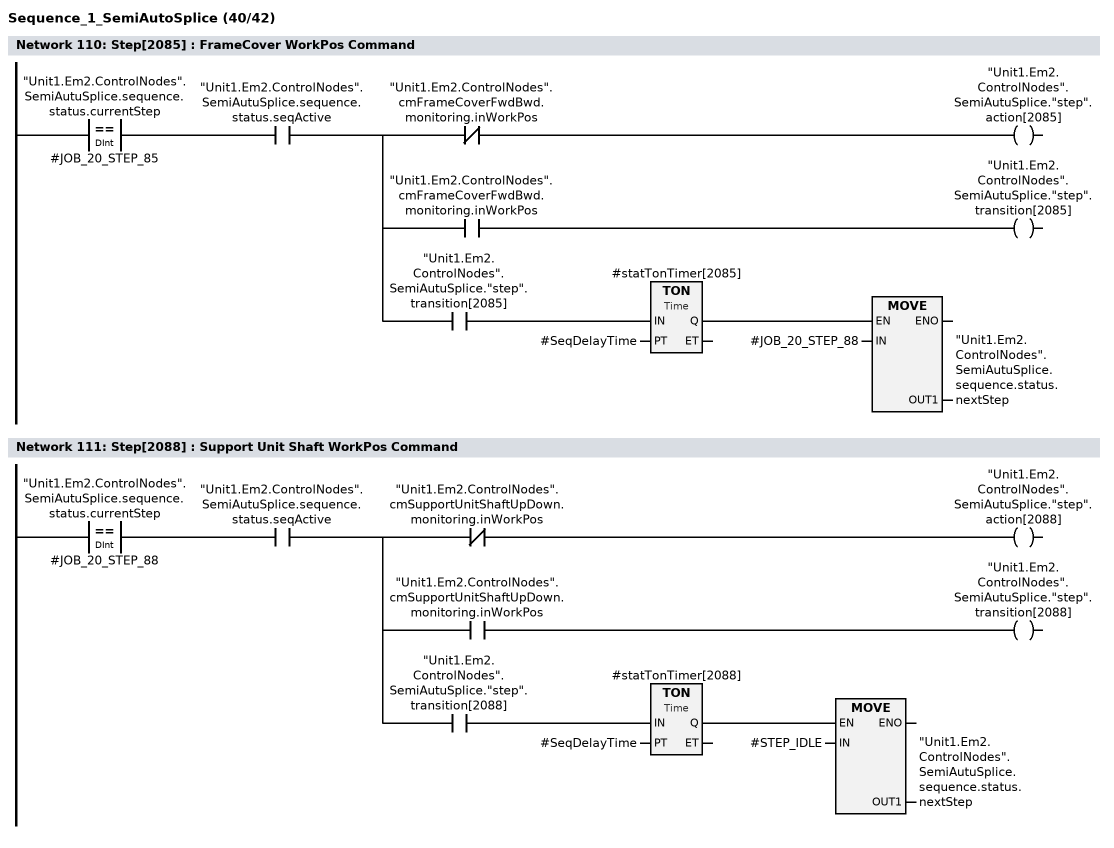
   RUNG wire#powerrail
      { S7_Templates := "SrcType := DInt" } EQ_Contact(in1 := "Unit1.Em2.ControlNodes".SemiAutuSplice.sequence.status.currentStep, in2 := #JOB_20_STEP_85)
      Contact( "Unit1.Em2.ControlNodes".SemiAutuSplice.sequence.status.seqActive )
      wire#w1
      I_Contact( "Unit1.Em2.ControlNodes".cmFrameCoverFwdBwd.monitoring.inWorkPos )
      Coil( "Unit1.Em2.ControlNodes".SemiAutuSplice."step".action[2085] )
   END_RUNG
   RUNG wire#w1
      Contact( "Unit1.Em2.ControlNodes".cmFrameCoverFwdBwd.monitoring.inWorkPos )
      Coil( "Unit1.Em2.ControlNodes".SemiAutuSplice."step".transition[2085] )
   END_RUNG
   RUNG wire#w1
      Contact( "Unit1.Em2.ControlNodes".SemiAutuSplice."step".transition[2085] )
      { S7_Templates := "time_type := Time" } #statTonTimer[2085].TON(pt := #SeqDelayTime, et =>)
      Move(in := #JOB_20_STEP_88, out1 => "Unit1.Em2.ControlNodes".SemiAutuSplice.sequence.status.nextStep)
   END_RUNG
   // the same network as SCL:
   #_w1 := ("Unit1.Em2.ControlNodes".SemiAutuSplice.sequence.status.currentStep = #JOB_20_STEP_85) AND "Unit1.Em2.ControlNodes".SemiAutuSplice.sequence.status.seqActive;
   "Unit1.Em2.ControlNodes".SemiAutuSplice."step".action[2085] := #_w1 AND NOT "Unit1.Em2.ControlNodes".cmFrameCoverFwdBwd.monitoring.inWorkPos;
   "Unit1.Em2.ControlNodes".SemiAutuSplice."step".transition[2085] := #_w1 AND "Unit1.Em2.ControlNodes".cmFrameCoverFwdBwd.monitoring.inWorkPos;
   #statTonTimer[2085].TON(IN := #_w1 AND "Unit1.Em2.ControlNodes".SemiAutuSplice."step".transition[2085],
                           PT := #SeqDelayTime);
   IF #statTonTimer[2085].Q THEN
       "Unit1.Em2.ControlNodes".SemiAutuSplice.sequence.status.nextStep := #JOB_20_STEP_88;
   END_IF;
END_REGION

REGION Network 111: Step[2088] : Support Unit Shaft WorkPos Command
   RUNG wire#powerrail
      { S7_Templates := "SrcType := DInt" } EQ_Contact(in1 := "Unit1.Em2.ControlNodes".SemiAutuSplice.sequence.status.currentStep, in2 := #JOB_20_STEP_88)
      Contact( "Unit1.Em2.ControlNodes".SemiAutuSplice.sequence.status.seqActive )
      wire#w1
      I_Contact( "Unit1.Em2.ControlNodes".cmSupportUnitShaftUpDown.monitoring.inWorkPos )
      Coil( "Unit1.Em2.ControlNodes".SemiAutuSplice."step".action[2088] )
   END_RUNG
   RUNG wire#w1
      Contact( "Unit1.Em2.ControlNodes".cmSupportUnitShaftUpDown.monitoring.inWorkPos )
      Coil( "Unit1.Em2.ControlNodes".SemiAutuSplice."step".transition[2088] )
   END_RUNG
   RUNG wire#w1
      Contact( "Unit1.Em2.ControlNodes".SemiAutuSplice."step".transition[2088] )
      { S7_Templates := "time_type := Time" } #statTonTimer[2088].TON(pt := #SeqDelayTime, et =>)
      Move(in := #STEP_IDLE, out1 => "Unit1.Em2.ControlNodes".SemiAutuSplice.sequence.status.nextStep)
   END_RUNG
   // the same network as SCL:
   #_w1 := ("Unit1.Em2.ControlNodes".SemiAutuSplice.sequence.status.currentStep = #JOB_20_STEP_88) AND "Unit1.Em2.ControlNodes".SemiAutuSplice.sequence.status.seqActive;
   "Unit1.Em2.ControlNodes".SemiAutuSplice."step".action[2088] := #_w1 AND NOT "Unit1.Em2.ControlNodes".cmSupportUnitShaftUpDown.monitoring.inWorkPos;
   "Unit1.Em2.ControlNodes".SemiAutuSplice."step".transition[2088] := #_w1 AND "Unit1.Em2.ControlNodes".cmSupportUnitShaftUpDown.monitoring.inWorkPos;
   #statTonTimer[2088].TON(IN := #_w1 AND "Unit1.Em2.ControlNodes".SemiAutuSplice."step".transition[2088],
                           PT := #SeqDelayTime);
   IF #statTonTimer[2088].Q THEN
       "Unit1.Em2.ControlNodes".SemiAutuSplice.sequence.status.nextStep := #STEP_IDLE;
   END_IF;
END_REGION

REGION Network 112: *************** IMMEDIATE STOP ****************
END_REGION

REGION Network 113: Immediate Stop
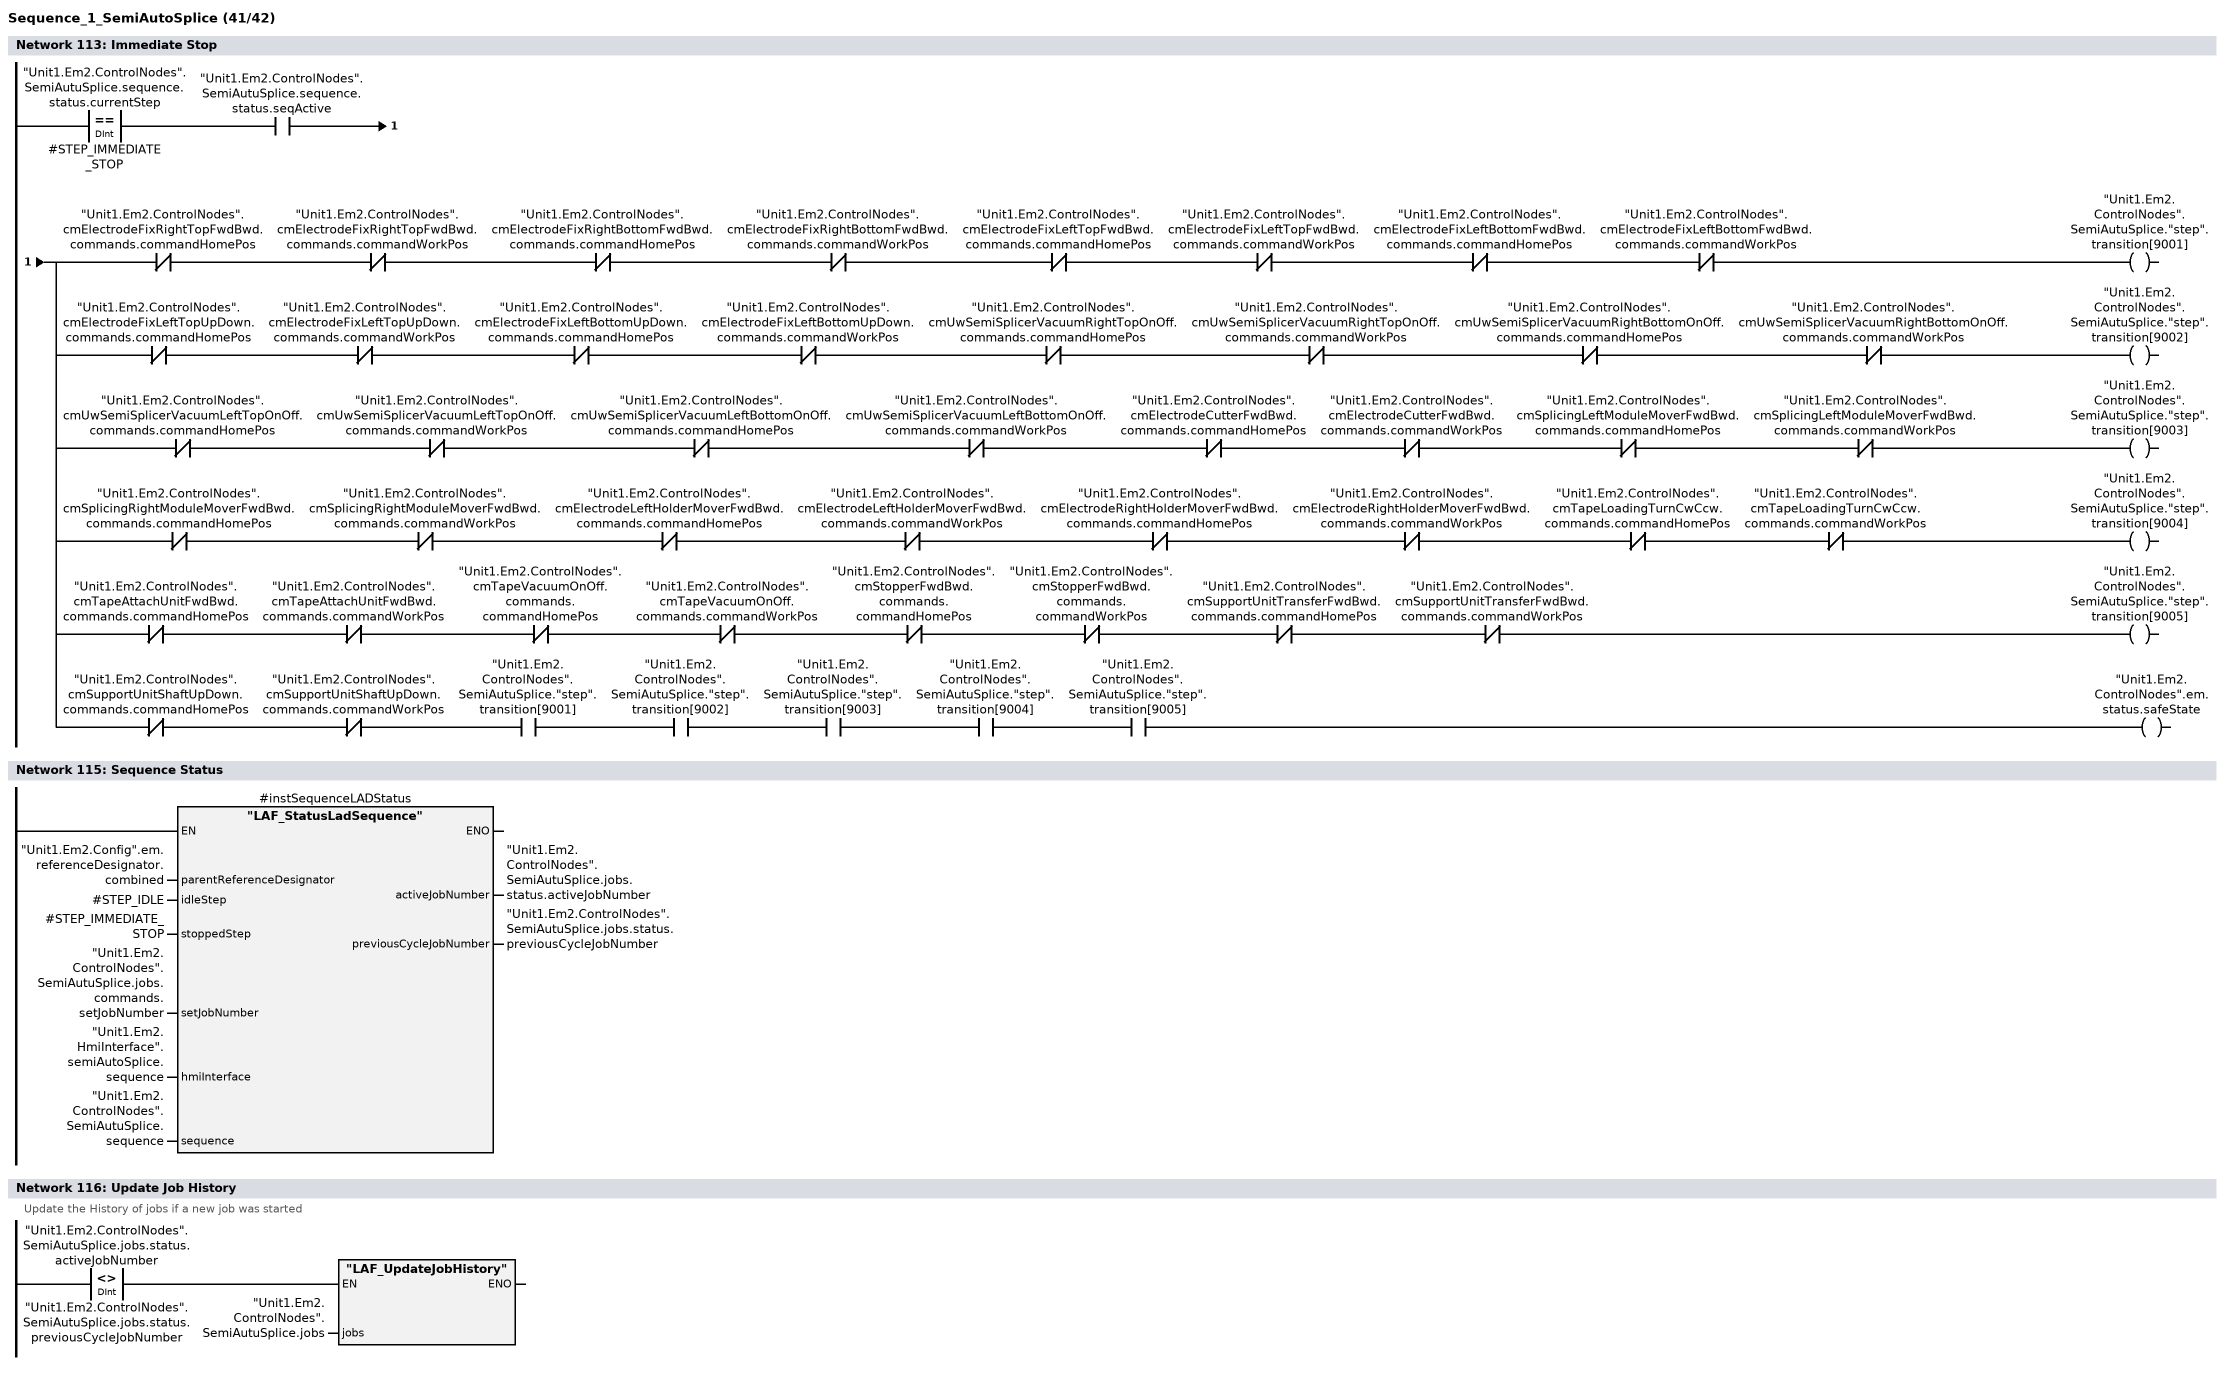
   RUNG wire#powerrail
      { S7_Templates := "SrcType := DInt" } EQ_Contact(in1 := "Unit1.Em2.ControlNodes".SemiAutuSplice.sequence.status.currentStep, in2 := #STEP_IMMEDIATE_STOP)
      Contact( "Unit1.Em2.ControlNodes".SemiAutuSplice.sequence.status.seqActive )
      wire#w1
      I_Contact( "Unit1.Em2.ControlNodes".cmElectrodeFixRightTopFwdBwd.commands.commandHomePos )
      I_Contact( "Unit1.Em2.ControlNodes".cmElectrodeFixRightTopFwdBwd.commands.commandWorkPos )
      I_Contact( "Unit1.Em2.ControlNodes".cmElectrodeFixRightBottomFwdBwd.commands.commandHomePos )
      I_Contact( "Unit1.Em2.ControlNodes".cmElectrodeFixRightBottomFwdBwd.commands.commandWorkPos )
      I_Contact( "Unit1.Em2.ControlNodes".cmElectrodeFixLeftTopFwdBwd.commands.commandHomePos )
      I_Contact( "Unit1.Em2.ControlNodes".cmElectrodeFixLeftTopFwdBwd.commands.commandWorkPos )
      I_Contact( "Unit1.Em2.ControlNodes".cmElectrodeFixLeftBottomFwdBwd.commands.commandHomePos )
      I_Contact( "Unit1.Em2.ControlNodes".cmElectrodeFixLeftBottomFwdBwd.commands.commandWorkPos )
      Coil( "Unit1.Em2.ControlNodes".SemiAutuSplice."step".transition[9001] )
   END_RUNG
   RUNG wire#w1
      I_Contact( "Unit1.Em2.ControlNodes".cmElectrodeFixLeftTopUpDown.commands.commandHomePos )
      I_Contact( "Unit1.Em2.ControlNodes".cmElectrodeFixLeftTopUpDown.commands.commandWorkPos )
      I_Contact( "Unit1.Em2.ControlNodes".cmElectrodeFixLeftBottomUpDown.commands.commandHomePos )
      I_Contact( "Unit1.Em2.ControlNodes".cmElectrodeFixLeftBottomUpDown.commands.commandWorkPos )
      I_Contact( "Unit1.Em2.ControlNodes".cmUwSemiSplicerVacuumRightTopOnOff.commands.commandHomePos )
      I_Contact( "Unit1.Em2.ControlNodes".cmUwSemiSplicerVacuumRightTopOnOff.commands.commandWorkPos )
      I_Contact( "Unit1.Em2.ControlNodes".cmUwSemiSplicerVacuumRightBottomOnOff.commands.commandHomePos )
      I_Contact( "Unit1.Em2.ControlNodes".cmUwSemiSplicerVacuumRightBottomOnOff.commands.commandWorkPos )
      Coil( "Unit1.Em2.ControlNodes".SemiAutuSplice."step".transition[9002] )
   END_RUNG
   RUNG wire#w1
      I_Contact( "Unit1.Em2.ControlNodes".cmUwSemiSplicerVacuumLeftTopOnOff.commands.commandHomePos )
      I_Contact( "Unit1.Em2.ControlNodes".cmUwSemiSplicerVacuumLeftTopOnOff.commands.commandWorkPos )
      I_Contact( "Unit1.Em2.ControlNodes".cmUwSemiSplicerVacuumLeftBottomOnOff.commands.commandHomePos )
      I_Contact( "Unit1.Em2.ControlNodes".cmUwSemiSplicerVacuumLeftBottomOnOff.commands.commandWorkPos )
      I_Contact( "Unit1.Em2.ControlNodes".cmElectrodeCutterFwdBwd.commands.commandHomePos )
      I_Contact( "Unit1.Em2.ControlNodes".cmElectrodeCutterFwdBwd.commands.commandWorkPos )
      I_Contact( "Unit1.Em2.ControlNodes".cmSplicingLeftModuleMoverFwdBwd.commands.commandHomePos )
      I_Contact( "Unit1.Em2.ControlNodes".cmSplicingLeftModuleMoverFwdBwd.commands.commandWorkPos )
      Coil( "Unit1.Em2.ControlNodes".SemiAutuSplice."step".transition[9003] )
   END_RUNG
   RUNG wire#w1
      I_Contact( "Unit1.Em2.ControlNodes".cmSplicingRightModuleMoverFwdBwd.commands.commandHomePos )
      I_Contact( "Unit1.Em2.ControlNodes".cmSplicingRightModuleMoverFwdBwd.commands.commandWorkPos )
      I_Contact( "Unit1.Em2.ControlNodes".cmElectrodeLeftHolderMoverFwdBwd.commands.commandHomePos )
      I_Contact( "Unit1.Em2.ControlNodes".cmElectrodeLeftHolderMoverFwdBwd.commands.commandWorkPos )
      I_Contact( "Unit1.Em2.ControlNodes".cmElectrodeRightHolderMoverFwdBwd.commands.commandHomePos )
      I_Contact( "Unit1.Em2.ControlNodes".cmElectrodeRightHolderMoverFwdBwd.commands.commandWorkPos )
      I_Contact( "Unit1.Em2.ControlNodes".cmTapeLoadingTurnCwCcw.commands.commandHomePos )
      I_Contact( "Unit1.Em2.ControlNodes".cmTapeLoadingTurnCwCcw.commands.commandWorkPos )
      Coil( "Unit1.Em2.ControlNodes".SemiAutuSplice."step".transition[9004] )
   END_RUNG
   RUNG wire#w1
      I_Contact( "Unit1.Em2.ControlNodes".cmTapeAttachUnitFwdBwd.commands.commandHomePos )
      I_Contact( "Unit1.Em2.ControlNodes".cmTapeAttachUnitFwdBwd.commands.commandWorkPos )
      I_Contact( "Unit1.Em2.ControlNodes".cmTapeVacuumOnOff.commands.commandHomePos )
      I_Contact( "Unit1.Em2.ControlNodes".cmTapeVacuumOnOff.commands.commandWorkPos )
      I_Contact( "Unit1.Em2.ControlNodes".cmStopperFwdBwd.commands.commandHomePos )
      I_Contact( "Unit1.Em2.ControlNodes".cmStopperFwdBwd.commands.commandWorkPos )
      I_Contact( "Unit1.Em2.ControlNodes".cmSupportUnitTransferFwdBwd.commands.commandHomePos )
      I_Contact( "Unit1.Em2.ControlNodes".cmSupportUnitTransferFwdBwd.commands.commandWorkPos )
      Coil( "Unit1.Em2.ControlNodes".SemiAutuSplice."step".transition[9005] )
   END_RUNG
   RUNG wire#w1
      I_Contact( "Unit1.Em2.ControlNodes".cmSupportUnitShaftUpDown.commands.commandHomePos )
      I_Contact( "Unit1.Em2.ControlNodes".cmSupportUnitShaftUpDown.commands.commandWorkPos )
      Contact( "Unit1.Em2.ControlNodes".SemiAutuSplice."step".transition[9001] )
      Contact( "Unit1.Em2.ControlNodes".SemiAutuSplice."step".transition[9002] )
      Contact( "Unit1.Em2.ControlNodes".SemiAutuSplice."step".transition[9003] )
      Contact( "Unit1.Em2.ControlNodes".SemiAutuSplice."step".transition[9004] )
      Contact( "Unit1.Em2.ControlNodes".SemiAutuSplice."step".transition[9005] )
      Coil( "Unit1.Em2.ControlNodes".em.status.safeState )
   END_RUNG
   // the same network as SCL:
   #_w1 := ("Unit1.Em2.ControlNodes".SemiAutuSplice.sequence.status.currentStep = #STEP_IMMEDIATE_STOP) AND "Unit1.Em2.ControlNodes".SemiAutuSplice.sequence.status.seqActive;
   "Unit1.Em2.ControlNodes".SemiAutuSplice."step".transition[9001] := #_w1 AND NOT "Unit1.Em2.ControlNodes".cmElectrodeFixRightTopFwdBwd.commands.commandHomePos AND NOT "Unit1.Em2.ControlNodes".cmElectrodeFixRightTopFwdBwd.commands.commandWorkPos AND NOT "Unit1.Em2.ControlNodes".cmElectrodeFixRightBottomFwdBwd.commands.commandHomePos AND NOT "Unit1.Em2.ControlNodes".cmElectrodeFixRightBottomFwdBwd.commands.commandWorkPos AND NOT "Unit1.Em2.ControlNodes".cmElectrodeFixLeftTopFwdBwd.commands.commandHomePos AND NOT "Unit1.Em2.ControlNodes".cmElectrodeFixLeftTopFwdBwd.commands.commandWorkPos AND NOT "Unit1.Em2.ControlNodes".cmElectrodeFixLeftBottomFwdBwd.commands.commandHomePos AND NOT "Unit1.Em2.ControlNodes".cmElectrodeFixLeftBottomFwdBwd.commands.commandWorkPos;
   "Unit1.Em2.ControlNodes".SemiAutuSplice."step".transition[9002] := #_w1 AND NOT "Unit1.Em2.ControlNodes".cmElectrodeFixLeftTopUpDown.commands.commandHomePos AND NOT "Unit1.Em2.ControlNodes".cmElectrodeFixLeftTopUpDown.commands.commandWorkPos AND NOT "Unit1.Em2.ControlNodes".cmElectrodeFixLeftBottomUpDown.commands.commandHomePos AND NOT "Unit1.Em2.ControlNodes".cmElectrodeFixLeftBottomUpDown.commands.commandWorkPos AND NOT "Unit1.Em2.ControlNodes".cmUwSemiSplicerVacuumRightTopOnOff.commands.commandHomePos AND NOT "Unit1.Em2.ControlNodes".cmUwSemiSplicerVacuumRightTopOnOff.commands.commandWorkPos AND NOT "Unit1.Em2.ControlNodes".cmUwSemiSplicerVacuumRightBottomOnOff.commands.commandHomePos AND NOT "Unit1.Em2.ControlNodes".cmUwSemiSplicerVacuumRightBottomOnOff.commands.commandWorkPos;
   "Unit1.Em2.ControlNodes".SemiAutuSplice."step".transition[9003] := #_w1 AND NOT "Unit1.Em2.ControlNodes".cmUwSemiSplicerVacuumLeftTopOnOff.commands.commandHomePos AND NOT "Unit1.Em2.ControlNodes".cmUwSemiSplicerVacuumLeftTopOnOff.commands.commandWorkPos AND NOT "Unit1.Em2.ControlNodes".cmUwSemiSplicerVacuumLeftBottomOnOff.commands.commandHomePos AND NOT "Unit1.Em2.ControlNodes".cmUwSemiSplicerVacuumLeftBottomOnOff.commands.commandWorkPos AND NOT "Unit1.Em2.ControlNodes".cmElectrodeCutterFwdBwd.commands.commandHomePos AND NOT "Unit1.Em2.ControlNodes".cmElectrodeCutterFwdBwd.commands.commandWorkPos AND NOT "Unit1.Em2.ControlNodes".cmSplicingLeftModuleMoverFwdBwd.commands.commandHomePos AND NOT "Unit1.Em2.ControlNodes".cmSplicingLeftModuleMoverFwdBwd.commands.commandWorkPos;
   "Unit1.Em2.ControlNodes".SemiAutuSplice."step".transition[9004] := #_w1 AND NOT "Unit1.Em2.ControlNodes".cmSplicingRightModuleMoverFwdBwd.commands.commandHomePos AND NOT "Unit1.Em2.ControlNodes".cmSplicingRightModuleMoverFwdBwd.commands.commandWorkPos AND NOT "Unit1.Em2.ControlNodes".cmElectrodeLeftHolderMoverFwdBwd.commands.commandHomePos AND NOT "Unit1.Em2.ControlNodes".cmElectrodeLeftHolderMoverFwdBwd.commands.commandWorkPos AND NOT "Unit1.Em2.ControlNodes".cmElectrodeRightHolderMoverFwdBwd.commands.commandHomePos AND NOT "Unit1.Em2.ControlNodes".cmElectrodeRightHolderMoverFwdBwd.commands.commandWorkPos AND NOT "Unit1.Em2.ControlNodes".cmTapeLoadingTurnCwCcw.commands.commandHomePos AND NOT "Unit1.Em2.ControlNodes".cmTapeLoadingTurnCwCcw.commands.commandWorkPos;
   "Unit1.Em2.ControlNodes".SemiAutuSplice."step".transition[9005] := #_w1 AND NOT "Unit1.Em2.ControlNodes".cmTapeAttachUnitFwdBwd.commands.commandHomePos AND NOT "Unit1.Em2.ControlNodes".cmTapeAttachUnitFwdBwd.commands.commandWorkPos AND NOT "Unit1.Em2.ControlNodes".cmTapeVacuumOnOff.commands.commandHomePos AND NOT "Unit1.Em2.ControlNodes".cmTapeVacuumOnOff.commands.commandWorkPos AND NOT "Unit1.Em2.ControlNodes".cmStopperFwdBwd.commands.commandHomePos AND NOT "Unit1.Em2.ControlNodes".cmStopperFwdBwd.commands.commandWorkPos AND NOT "Unit1.Em2.ControlNodes".cmSupportUnitTransferFwdBwd.commands.commandHomePos AND NOT "Unit1.Em2.ControlNodes".cmSupportUnitTransferFwdBwd.commands.commandWorkPos;
   "Unit1.Em2.ControlNodes".em.status.safeState := #_w1 AND NOT "Unit1.Em2.ControlNodes".cmSupportUnitShaftUpDown.commands.commandHomePos AND NOT "Unit1.Em2.ControlNodes".cmSupportUnitShaftUpDown.commands.commandWorkPos AND "Unit1.Em2.ControlNodes".SemiAutuSplice."step".transition[9001] AND "Unit1.Em2.ControlNodes".SemiAutuSplice."step".transition[9002] AND "Unit1.Em2.ControlNodes".SemiAutuSplice."step".transition[9003] AND "Unit1.Em2.ControlNodes".SemiAutuSplice."step".transition[9004] AND "Unit1.Em2.ControlNodes".SemiAutuSplice."step".transition[9005];
END_REGION

REGION Network 114: *************** STATUS **********************
END_REGION

REGION Network 115: Sequence Status
   RUNG wire#powerrail
      #instSequenceLADStatus(parentReferenceDesignator := "Unit1.Em2.Config".em.referenceDesignator.combined, idleStep := #STEP_IDLE, stoppedStep := #STEP_IMMEDIATE_STOP, setJobNumber := "Unit1.Em2.ControlNodes".SemiAutuSplice.jobs.commands.setJobNumber, hmiInterface := "Unit1.Em2.HmiInterface".semiAutoSplice.sequence, sequence := "Unit1.Em2.ControlNodes".SemiAutuSplice.sequence, activeJobNumber => "Unit1.Em2.ControlNodes".SemiAutuSplice.jobs.status.activeJobNumber, previousCycleJobNumber => "Unit1.Em2.ControlNodes".SemiAutuSplice.jobs.status.previousCycleJobNumber)
   END_RUNG
   // the same network as SCL:
   #instSequenceLADStatus(parentReferenceDesignator := "Unit1.Em2.Config".em.referenceDesignator.combined,   // "LAF_StatusLadSequence"
                          idleStep := #STEP_IDLE,
                          stoppedStep := #STEP_IMMEDIATE_STOP,
                          setJobNumber := "Unit1.Em2.ControlNodes".SemiAutuSplice.jobs.commands.setJobNumber,
                          hmiInterface := "Unit1.Em2.HmiInterface".semiAutoSplice.sequence,
                          sequence := "Unit1.Em2.ControlNodes".SemiAutuSplice.sequence,
                          activeJobNumber => "Unit1.Em2.ControlNodes".SemiAutuSplice.jobs.status.activeJobNumber,
                          previousCycleJobNumber => "Unit1.Em2.ControlNodes".SemiAutuSplice.jobs.status.previousCycleJobNumber);
END_REGION

REGION Network 116: Update Job History
   // Update the History of jobs if a new job was started
   RUNG wire#powerrail
      { S7_Templates := "SrcType := DInt" } NE_Contact(in1 := "Unit1.Em2.ControlNodes".SemiAutuSplice.jobs.status.activeJobNumber, in2 := "Unit1.Em2.ControlNodes".SemiAutuSplice.jobs.status.previousCycleJobNumber)
      "LAF_UpdateJobHistory"(jobs := "Unit1.Em2.ControlNodes".SemiAutuSplice.jobs)
   END_RUNG
   // the same network as SCL:
   IF "Unit1.Em2.ControlNodes".SemiAutuSplice.jobs.status.activeJobNumber <> "Unit1.Em2.ControlNodes".SemiAutuSplice.jobs.status.previousCycleJobNumber THEN
       "LAF_UpdateJobHistory"(jobs := "Unit1.Em2.ControlNodes".SemiAutuSplice.jobs);
   END_IF;
END_REGION

REGION Network 117: Output steps as String
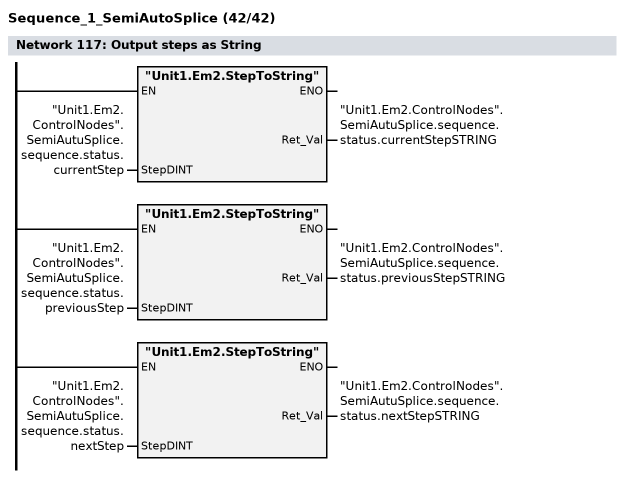
   RUNG wire#powerrail
      "Unit1.Em2.StepToString"(StepDINT := "Unit1.Em2.ControlNodes".SemiAutuSplice.sequence.status.currentStep, Ret_Val => "Unit1.Em2.ControlNodes".SemiAutuSplice.sequence.status.currentStepSTRING)
   END_RUNG
   RUNG wire#powerrail
      "Unit1.Em2.StepToString"(StepDINT := "Unit1.Em2.ControlNodes".SemiAutuSplice.sequence.status.previousStep, Ret_Val => "Unit1.Em2.ControlNodes".SemiAutuSplice.sequence.status.previousStepSTRING)
   END_RUNG
   RUNG wire#powerrail
      "Unit1.Em2.StepToString"(StepDINT := "Unit1.Em2.ControlNodes".SemiAutuSplice.sequence.status.nextStep, Ret_Val => "Unit1.Em2.ControlNodes".SemiAutuSplice.sequence.status.nextStepSTRING)
   END_RUNG
   // the same network as SCL:
   "Unit1.Em2.ControlNodes".SemiAutuSplice.sequence.status.currentStepSTRING := "Unit1.Em2.StepToString"(StepDINT := "Unit1.Em2.ControlNodes".SemiAutuSplice.sequence.status.currentStep);
   "Unit1.Em2.ControlNodes".SemiAutuSplice.sequence.status.previousStepSTRING := "Unit1.Em2.StepToString"(StepDINT := "Unit1.Em2.ControlNodes".SemiAutuSplice.sequence.status.previousStep);
   "Unit1.Em2.ControlNodes".SemiAutuSplice.sequence.status.nextStepSTRING := "Unit1.Em2.StepToString"(StepDINT := "Unit1.Em2.ControlNodes".SemiAutuSplice.sequence.status.nextStep);
END_REGION
END_FUNCTION_BLOCK
